{attribute addProperty BoxType "EL6695-0002-0001"}
{attribute addProperty Id "SYNC_InputsAT %I*SYNC_Inputs_45196B502430IO_InputsEMPTY_STRUCTURE000IO_OutputsEMPTY_STRUCTURE000WcStateAT %I*WcState_F855686C1620InfoDataAT %I*InfoData_275E3363128160"}
{attribute addProperty CRC "3482193852"}
{attribute addProperty SizeInBites "168"}
{attribute addProperty SizeInBytes "21"}
TYPE EL6695_952642F6 :
STRUCT
	{attribute addProperty Name "SYNC_Inputs"}
	SYNC_Inputs : SYNC_Inputs_45196B50;
	{attribute addProperty Name "IO_Inputs"}
	IO_Inputs : EMPTY_STRUCTURE;
	{attribute addProperty Name "IO_Outputs"}
	IO_Outputs : EMPTY_STRUCTURE;
	{attribute addProperty Name "WcState"}
	WcState : WcState_F855686C;
	{attribute addProperty Name "InfoData"}
	InfoData : InfoData_275E3363;
END_STRUCT
END_TYPE

(* stored: Version 1.2.0.0, ProductVersion 3.1.4024.9
   DUT EL6695_952642F6: Id {c40fb80e-81d8-4abc-af58-f6a0aeb89a2e} *)
